INTERFACE I_Color

PROPERTY Alpha : BYTE
GET
END_GET
SET
END_SET
END_PROPERTY

PROPERTY Blue : BYTE
GET
END_GET
SET
END_SET
END_PROPERTY

METHOD Clone
VAR_INPUT
	iColor	: I_Color;
END_VAR
END_METHOD

PROPERTY Green : BYTE
GET
END_GET
SET
END_SET
END_PROPERTY

PROPERTY Raw : DWORD
GET
END_GET
SET
END_SET
END_PROPERTY

PROPERTY Red : BYTE
GET
END_GET
SET
END_SET
END_PROPERTY

METHOD Set
VAR_INPUT
	nRed: USINT;
	nGreen: USINT;
	nBlue: USINT;
	nAlpha: USINT;
END_VAR
END_METHOD

END_INTERFACE

(* stored: Version 1.1.0.1
   Itf I_Color: Id {c14a9189-f87c-457b-89d1-843d3ff3e927}
   Property Alpha: Id {dbf4dd98-9843-49d4-a908-5b54536c0014}
   Get Get: Id {9125f2f4-4319-42f5-bd1c-7acf4a5f281f}
   Set Set: Id {d8a83b14-fb5a-47e8-9536-c3c50ce9ca55}
   Property Blue: Id {573c36d9-70a0-4842-aedd-2c0046f57d09}
   Get Get: Id {95cdea63-da39-4e73-b37a-2cd660b4715f}
   Set Set: Id {94859b13-b99b-4fcd-8dc9-709951bc754b}
   Method Clone: Id {f4bbf03f-d112-42dc-9b12-ed0c9fde6c5b}
   Property Green: Id {ab9240df-3a6b-48c6-8fe8-51f28a6799ac}
   Get Get: Id {2e3600d0-684c-4c70-8b84-5c271cc4941e}
   Set Set: Id {c2b4d1e8-024b-4a08-91a0-33591d5f27fe}
   Property Raw: Id {71a4be24-f240-4748-875e-15491da3629e}
   Get Get: Id {9aede787-8993-471e-992b-ce11ca65f74b}
   Set Set: Id {96b67c65-e940-4056-8367-d2bb4c000729}
   Property Red: Id {8f5f31c6-f487-4b41-8b3c-de67989885fa}
   Get Get: Id {e0520e32-cff6-456b-adee-36addba7abca}
   Set Set: Id {a7ed6ac8-2d10-4865-9796-07711d52c419}
   Method Set: Id {d14e615a-60bc-4338-b82b-982841ae87b8} *)
